Staubli VAL3: onF8Event.pgx

program onF8Event(bool& x_bExit[])
  local string l_sMessage
  local string l_sButton[2]
  local num l_nIndex
  local string l_sEvent
  local num l_nKey
begin
  // look if the bButton is enable

end
